GLOBALCONSTANTS sequence (* Global constants *)
  (* Standard: 61499-1; Description: Copyright (c) 2024 HR Agrartechnik GmbH This program and the accompanying materials are made available under the terms of the Eclipse Public License 2.0 which is available at https://www.eclipse.org/legal/epl-2.0/ SPDX-License-Identifier: EPL-2.0 *)
  (* Version 1.0, 2024-03-02, Franz Höpfinger, HR Agrartechnik GmbH *)
  VAR_GLOBAL CONSTANT
    NO_TIME : TIME := TIME#49d17h2m47s295ms;
    State_00 : SINT := SINT#0;
    State_01 : SINT := SINT#1;
    State_02 : SINT := SINT#2;
    State_03 : SINT := SINT#3;
    State_04 : SINT := SINT#4;
    State_05 : SINT := SINT#5;
    State_06 : SINT := SINT#6;
    State_07 : SINT := SINT#7;
    State_08 : SINT := SINT#8;
  END_VAR
END_GLOBALCONSTANTS
